KUKA KRL program: Main.src, Main.dat

--- Main.src ---
&ACCESS RVP
&REL 6
DEF Main()

GLOBAL INTERRUPT DECL 3 WHEN $STOPMESS==True DO IR_STOPM()
INTERRUPT ON 3
BAS(#INITMOV,0)

DECL INT Cmd
DECL INT OvSave

;Robot_Cmd_RoutineID   from PLC   0 = idle, anything else = run that routine
;Robot_Sts_State       to PLC     0 idle   1 running   2 done   3 faulted
;Robot_Sts_RoutineID   to PLC     echo of the routine being run
;
;10 Home          20 UpStacker    30 LaserMarker   40 IMM
;50 SprueCutter   60 DownStacker  71 72 73 Reject blank / finished / both

BeginningOfModule:
RobotCell_Error=False
RtoPLC_RobotReachedStop=False
Robot_Sts_State=0
Robot_Sts_RoutineID=0

OvSave=$OV_PRO
$OV_PRO=30
GoHome()
$OV_PRO=OvSave

RtoIMM_RobotWithIMM=True
RtoIMM_MoldAreaFree=True
RtoIMM_MoldCloseEnable=True
RtoIMM_MoldOpenEnable=True
RtoPLC_ToolBlnkMrked=False


Loop

If ((PLCtoR_Stop==True) Or (PLCtoR_DrawerInPos==False)) Then
   GoHome()
   RtoIMM_MoldAreaFree=True
   RtoIMM_MoldCloseEnable=True
   RtoIMM_MoldOpenEnable=True
   Robot_Sts_State=0
   Robot_Sts_RoutineID=0
   RtoPLC_RobotReachedStop=True
   Wait for $EXT_START
   RtoPLC_RobotReachedStop=False
EndIf

Wait for ((Robot_Cmd_RoutineID<>0) Or (PLCtoR_Stop==True) Or (PLCtoR_DrawerInPos==False))

If Robot_Cmd_RoutineID<>0 Then

   Cmd=Robot_Cmd_RoutineID
   Robot_Sts_RoutineID=Cmd
   Robot_Sts_State=1

   Switch Cmd
   Case 10
      GoHome()
   Case 20
      Station200_UpStacker()
   Case 30
      Station300_LaserMarker()
   Case 40
      Station400_IMM()
   Case 50
      Station500_SprueCutter()
   Case 60
      Station600_DownStacker()
   Case 71,72,73
      Rjct_1Blnk_2Fin_3Both=Cmd-70
      Station500_Reject()
   Default
      RobotCell_Error=True
   EndSwitch

   If RobotCell_Error==True Then
      Robot_Sts_State=3
   Else
      Robot_Sts_State=2
   EndIf

   Wait for Robot_Cmd_RoutineID==0

   If RobotCell_Error==True Then
      GOTO BeginningOfModule
   EndIf

   Robot_Sts_State=0
   Robot_Sts_RoutineID=0

EndIf

EndLoop
END


DEF GoHome()
PDAT_ACT=PDEFAULT
FDAT_ACT=FHOME
BAS(#PTP_PARAMS,100)
$H_POS=XHOME
PTP XHOME
END

--- Main.dat ---
DEFDAT Main
   ;FOLD EXTERNAL DECLARATIONS;%{PE}%MKUKATPBASIS,%CEXT,%VCOMMON,%P
   ;FOLD BASISTECH EXT;%{PE}%MKUKATPBASIS,%CEXT,%VEXT,%P
   EXT BAS(BAS_COMMAND :IN, REAL :IN)
   DECL INT SUCCESS
   ;ENDFOLD (BASISTECH EXT)
   ;FOLD USER EXT;%{E}%MKUKATPUSER,%CEXT,%VEXT,%P
   ;Make your modifications here

   ;ENDFOLD (USER EXT)
   ;ENDFOLD (EXTERNAL DECLARATIONS)
   ; Local PDEFAULT, copied verbatim from the previous Main.dat.
   ;
   ; This file exists ONLY for this declaration. $config.dat also declares a
   ; global PDEFAULT, but with ACC 100.000. A module-local declaration shadows
   ; the global, so the old Main has always used ACC 35.000. Ship Main.src
   ; without this .dat and every home move silently runs at roughly three
   ; times the joint acceleration it does today.
   DECL PDAT PDEFAULT = { APO_MODE #CDIS, APO_DIST 500.0, VEL 100.0, ACC 35.000, GEAR_JERK 100.0, EXAX_IGN 0 }
ENDDAT
